TYPE INT_LENGTH : INT(0..32767); END_TYPE

(* stored: Version 1.1.0.1
   DUT INT_LENGTH: Id {a781777b-a6c5-4629-bcf2-ce9e17dd7dc7} *)
